// TIA Portal V20 export
VAR_GLOBAL   // PLC tag table "Unit1Em6_Servo"
   "BA040AZSBK17.00" AT %I1064.0 : Bool;   // FINAL ROLLER FRONT LIMIT SENSOR(-)
   "BA040AZSBK17.01" AT %I1064.1 : Bool;   // FINAL ROLLER FRONT HOME SENSOR
   "BA040AZSBK17.02" AT %I1064.2 : Bool;   // FINAL ROLLER FRONT LIMIT SENSOR(+)
   "BA040AZSBK17.04" AT %I1064.4 : Bool;   // FINAL ROLLER REAR LIMIT SENSOR(-)
   "BA040AZSBK17.05" AT %I1064.5 : Bool;   // FINAL ROLLER REAR HOME SENSOR
   "BA040AZSBK17.06" AT %I1064.6 : Bool;   // FINAL ROLLER REAR LIMIT SENSOR(+)
   "BA040AZSBK18.00" AT %I1068.0 : Bool;   // ANODE MANDREL REAR Y AXIS LIMIT SENSOR(-)
   "BA040AZSBK18.01" AT %I1068.1 : Bool;   // ANODE MANDREL REAR Y AXIS LIMIT SENSOR(+)
   "BA040AZSBK18.02" AT %I1068.2 : Bool;   // ANODE MANDREL REAR Z AXIS LIMIT SENSOR(-)
   "BA040AZSBK18.03" AT %I1068.3 : Bool;   // ANODE MANDREL REAR Z AXIS LIMIT SENSOR(+)
   "BA040AZSBK18.04" AT %I1068.4 : Bool;   // ANODE MANDREL FRONT Y AXIS LIMIT SENSOR(-)
   "BA040AZSBK18.05" AT %I1068.5 : Bool;   // ANODE MANDREL FRONT Y AXIS LIMIT SENSOR(+)
   "BA040AZSBK18.06" AT %I1068.6 : Bool;   // ANODE MANDREL FRONT Z AXIS LIMIT SENSOR(-)
   "BA040AZSBK18.07" AT %I1068.7 : Bool;   // ANODE MANDREL FRONT Z AXIS LIMIT SENSOR(+)
   "BA040AZSBK18.10" AT %I1069.0 : Bool;   // ANODE MANDREL REAR Y AXIS HOME SENSOR
   "BA040AZSBK18.12" AT %I1069.2 : Bool;   // ANODE MANDREL REAR Z AXIS HOME SENSOR
   "BA040AZSBK18.14" AT %I1069.4 : Bool;   // ANODE MANDREL FRONT Y AXIS HOME SENSOR
   "BA040AZSBK18.16" AT %I1069.6 : Bool;   // ANODE MANDREL FRONT Z AXIS HOME SENSOR
   "BA040AZSBK19.00" AT %I1072.0 : Bool;   // CATHODE MANDREL REAR Y AXIS LIMIT SENSOR(-)
   "BA040AZSBK19.01" AT %I1072.1 : Bool;   // CATHODE MANDREL REAR Y AXIS LIMIT SENSOR(+)
   "BA040AZSBK19.02" AT %I1072.2 : Bool;   // CATHODE MANDREL REAR Z AXIS LIMIT SENSOR(-)
   "BA040AZSBK19.03" AT %I1072.3 : Bool;   // CATHODE MANDREL REAR Z AXIS LIMIT SENSOR(+)
   "BA040AZSBK19.04" AT %I1072.4 : Bool;   // CATHODE MANDREL FRONT Y AXIS LIMIT SENSOR(-)
   "BA040AZSBK19.05" AT %I1072.5 : Bool;   // CATHODE MANDREL FRONT Y AXIS LIMIT SENSOR(+)
   "BA040AZSBK19.06" AT %I1072.6 : Bool;   // CATHODE MANDREL FRONT Z AXIS LIMIT SENSOR(-)
   "BA040AZSBK19.07" AT %I1072.7 : Bool;   // CATHODE MANDREL FRONT Z AXIS LIMIT SENSOR(+)
   "BA040AZSBK19.10" AT %I1073.0 : Bool;   // CATHODE MANDREL REAR Y AXIS HOME SENSOR
   "BA040AZSBK19.12" AT %I1073.2 : Bool;   // CATHODE MANDREL REAR Z AXIS HOME SENSOR
   "BA040AZSBK19.14" AT %I1073.4 : Bool;   // CATHODE MANDREL FRONT Y AXIS HOME SENSOR
   "BA040AZSBK19.16" AT %I1073.6 : Bool;   // CATHODE MANDREL FRONT Z AXIS HOME SENSOR
   "BA040AZSBK20.00" AT %I1076.0 : Bool;   // STACK TABLE Z-AXIS LIMIT SENSOR(-)
   "BA040AZSBK20.01" AT %I1076.1 : Bool;   // STACK TABLE Z-AXIS LIMIT SENSOR(+)
   "BA040AZSBK20.04" AT %I1076.4 : Bool;   // STACK TABLE OUT FRONT Z-AXIS LIMIT SENSOR(-)
   "BA040AZSBK20.05" AT %I1076.5 : Bool;   // STACK TABLE OUT FRONT Z-AXIS LIMIT SENSOR(+)
   "BA040AZSBK20.10" AT %I1077.0 : Bool;   // STACK TABLE Z-AXIS HOME SENSOR
   "BA040AZSBK20.14" AT %I1077.4 : Bool;   // STACK TABLE OUT FRONT Z-AXIS HOME SENSOR
   "BA040AZSBK14.01" AT %I1052.1 : Bool;   // STACK TABLE OUT REAR Z-AXIS LIMIT SENSOR(-)
   "BA040AZSBK14.03" AT %I1052.3 : Bool;   // STACK TABLE OUT REAR Z-AXIS LIMIT SENSOR(+)
   "BA040AZSBK14.11" AT %I1053.1 : Bool;   // STACK TABLE OUT REAR Z-AXIS HOME SENSOR
END_VAR
